PROGRAM MachineSimulation
VAR
	fbMachine	:	FB_MachineSimulator;
	
	i_SimReqBP	AT	%I*	:	ST_BeamParams;
	q_SimCurrBP	AT %Q*	:	ST_BeamParams;
END_VAR

//Machine simulator
fbMachine(
	i_stAssertedParams := i_SimReqBP,
	q_stMachineParams => PMPS_GVL_BeamParams.stCurrentBeamParameters,
	i_xFault	:= NOT GVL.g_FastFaultOutput1.q_xFastFaultOut
	);
	
q_SimCurrBP	:= fbMachine.q_stMachineParams;
q_SimCurrBP.neVReqRange := i_SimReqBP.neVReqRange;

END_PROGRAM

(* stored: Version 1.1.0.1, ProductVersion 3.1.4022.12
   POU MachineSimulation: Id {215532fb-b2c1-07b9-12dd-bf8b9df2fcb5}, SpecialFunc None *)
